FUNCTION alg_M_example_controller_pickpos : ARRAY[0..3] OF DINT
VAR_INPUT
	state: STATE;
END_VAR

alg_M_example_controller_pickpos := makeArray0(0, 1, 0, 2);

END_FUNCTION

(* stored: Version 1.1.0.1, ProductVersion 3.1.4022.18
   POU alg_M_example_controller_pickpos: Id {a7b73084-3338-4150-bcd2-b695d2757b38}, SpecialFunc None *)
